KUKA KRL program: chk_w4_grp3_opn.src

&ACCESS RVO2
&REL 7
&COMMENT Check GRP Z3 ACCELO OPEN
DEF chk_w4_grp3_opn( )

; Check gripper accelo OPEN Z3.1/2/3/4/5
;//---- Start User-------

$TIMER[10] = 0
$TIMER_STOP[10] = FALSE

WAIT FOR (NOT $IN[50] AND NOT $IN[52])
WAIT FOR ($IN[49] AND $IN[51])

$TIMER_STOP[10] = TRUE
$TIMER[10] = 0

;//---- End User---------

END
